FUNCTION_BLOCK IN_ARRAY (* ARRAY input from TextField-see IN_ANY *)
  (* Standard: 61499-1; Classification: GUI *)
  (* Version 0.0, 2000-04-19, JHC, Rockwell Automation *)
  (* Compiler header: package fb.rt.hmi; import java.awt.*; *)
  (* Compiler classdef: public class IN_ARRAY extends IN_ANY *)
  (* Compiler Java IBM VisualAge 3.0 *)
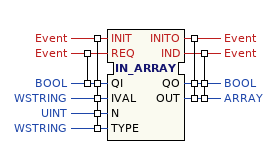
  EVENT_INPUT
    INIT WITH QI, IVAL, N, TYPE;
    REQ WITH QI;
  END_EVENT
  EVENT_OUTPUT
    INITO WITH QO, OUT;
    IND WITH QO, OUT;
  END_EVENT
  VAR_INPUT
    QI : BOOL;
    IVAL : WSTRING := "[]";
    N : UINT; (* Number of array elements *)
    TYPE : WSTRING; (* Array element type *)
  END_VAR
  VAR_OUTPUT
    QO : BOOL; (* 1=OK,0=Error *)
    OUT : ARRAY;
  END_VAR
END_FUNCTION_BLOCK
